// Mitsubishi GX Works2 project: pump_chem_up_NEW   PLC: FX3U/FX3UC

PROGRAM MAIN
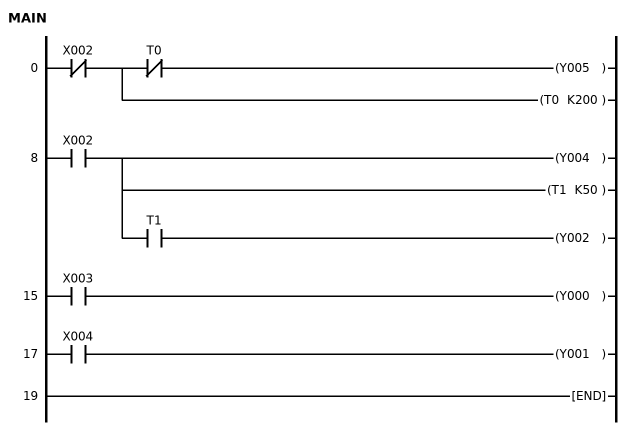
0     LDI     X002
      MPS
      ANI     T0
      OUT     Y005
      MPP
      OUT     T0 K200
8     LD      X002
      OUT     Y004
      OUT     T1 K50
      AND     T1
      OUT     Y002
15    LD      X003
      OUT     Y000
17    LD      X004
      OUT     Y001
19    END
END_PROGRAM
